// TIA Portal V20 export
// export: Created 2025-09-17T11:53:00.0000000Z, ExportSetting WithDefaults
ORGANIZATION_BLOCK "OB1_Main"   // OB1, SCL
TITLE = Main Program [OB1]
AUTHOR : Jules
VERSION : 0.1
// Main program block for the AHU Controller. Contains all I/O mapping, control logic, and FB calls.
// stored: AutoNumber false, IsOptimized true
BEGIN
   REGION INPUT MAPPING 
   (/**/) "IDB_SupplyFan".UDT.Run_Fdbk_DI := "AHU1_SF_RunFdbk";
   "IDB_SupplyFan".UDT.Airflow_Status_DI := "AHU1_SF_AirflowSw";
   "IDB_SupplyFan".UDT.VFD_Fault_DI := "AHU1_SF_VfdFault";
   "IDB_Cooling".UDT.CHW_Freeze_Stat_DI := "AHU1_CW_FreezeStat";
   "IDB_Cooling".UDT.CHW_Valve_Fdbk_AI := "AHU1_CW_VlvFdbk";
   "IDB_Heating".UDT.HW_Freeze_Stat_DI := "AHU1_HW_FreezeStat";
   "IDB_Heating".UDT.HW_Valve_Fdbk_AI := "AHU1_HW_VlvFdbk";
   "IDB_Damper".UDT.Return_Air_Temp_AI := "AHU1_RAT_Temp";
   "IDB_Damper".UDT.Outside_Air_Temp_AI := "AHU1_OAT_Temp";
   "IDB_Damper".UDT.Discharge_Air_Temp_AI := "AHU1_DAT_Temp";
   "IDB_Damper".UDT.Damper_Pos_Fdbk_AI := "AHU1_DMP_PosFdbk";
   "IDB_Monitoring".UDT.Dirty_Filter_DI := "AHU1_SYS_DirtyFilter";
   END_REGION

   REGION MAIN CONTROL LOGIC 
   (/**/) (/**/) (/**/) (/**/) (/**/) (/**/) (/**/) (/**/) (/**/) (/**/) (/**/) (/**/) (/**/) (/**/)END_REGION

   REGION FUNCTION BLOCK CALLS 
   (/**/) "IDB_SupplyFan"(Enable:= TRUE);(/**/) "IDB_Cooling"(Enable:= TRUE, Valve_Demand_In:= 0.0);(/**/) "IDB_Heating"(Enable:= TRUE, Valve_Demand_In:= 0.0);(/**/) "IDB_Damper"(Enable:= TRUE);
   "IDB_Monitoring"(Enable:= TRUE);
   END_REGION

   REGION OUTPUT MAPPING 
   (/**/) "AHU1_SF_StartCmd" := "IDB_SupplyFan".UDT.Start_Cmd_DO;
   "AHU1_SF_SpeedRef" := "IDB_SupplyFan".UDT.Speed_Ref_AO;
   "AHU1_CW_VlvCmd" := "IDB_Cooling".UDT.CHW_Valve_Cmd_AO;
   "AHU1_HW_VlvCmd" := "IDB_Heating".UDT.HW_Valve_Cmd_AO;
   "AHU1_DMP_PosCmd" := "IDB_Damper".UDT.Damper_Pos_Cmd_AO;
   END_REGION
END_ORGANIZATION_BLOCK
